(* PLC project Unnamed, Unknown Unnamed 1 *)
(* stored: creationDateTime 2024-12-03T22:58:12, modificationDateTime 2024-12-03T22:58:12 *)

CONFIGURATION Config0
  RESOURCE Res0 ON PLC
  END_RESOURCE
END_CONFIGURATION
